TYPE ST_GCSpinAxisMoveVelStatus EXTENDS ST_ServiceStatusBase :
STRUCT
	ActVel	: LREAL;
END_STRUCT
END_TYPE

(* stored: Version 1.1.0.1, ProductVersion 3.1.4026.18
   DUT ST_GCSpinAxisMoveVelStatus: Id {6c0d2dda-f2df-473a-8d9d-102f2eb1424e} *)
